(* IEC 61131-3 sources: Word/plc-course/12-data-structures/labs/starter, 3 files *)

(* ---- 12-1-recipe-manager.st ---- *)
(* Lab 12-1: Recipe manager - an array of structures, validated before use.
   Module 12 (Data structures). STARTER - the types, the recipe book, the
   limits and the program interface are declared for you. Write:
     1. the live check of the selected slot (SelectedOk),
     2. the load command: validate, then copy the whole recipe into Active,
        or reject it with the right LoadResult and change nothing.
   A FUNCTION for the value checks is a good idea (see the hint in the README).
   Then run:
     python3 tools/plctest.py 12-data-structures/labs/starter/12-1-recipe-manager.st *)

TYPE
  ST_Recipe :
  STRUCT
    Name    : STRING;               (* product name shown on the HMI; '' = empty slot *)
    Dose    : ARRAY[1..3] OF REAL;  (* kg of ingredient 1 (water), 2 (base), 3 (seasoning) *)
    Temp    : REAL;                 (* degC, batch temperature setpoint *)
    MixTime : TIME;                 (* mixing time once the batch is at temperature *)
  END_STRUCT;

  ST_RecipeLimits :
  STRUCT
    DoseMax    : REAL;              (* kg, largest dose of any one ingredient *)
    TotalMax   : REAL;              (* kg, vessel working capacity *)
    TempMin    : REAL;              (* degC *)
    TempMax    : REAL;              (* degC *)
    MixTimeMin : TIME;
    MixTimeMax : TIME;
  END_STRUCT;

  (* Result of the last load command. The first value is the initial value. *)
  E_LoadResult : (NotLoaded, Loaded, BadIndex, EmptySlot, BadValue, BatchBusy);
END_TYPE

PROGRAM RecipeManager
  VAR (* recipe book, edited on the HMI recipe screen. Slot 4 holds a typing
         mistake (95 degC) and slot 5 is empty, so both must be refused. *)
    Recipes : ARRAY[1..5] OF ST_Recipe := [
      (Name := 'Tomato soup',     Dose := [400.0, 150.0, 20.0], Temp := 85.0, MixTime := T#20m),
      (Name := 'Vegetable stock', Dose := [450.0, 300.0, 10.0], Temp := 80.0, MixTime := T#30m),
      (Name := 'Cheese sauce',    Dose := [250.0, 200.0, 50.0], Temp := 65.0, MixTime := T#15m),
      (Name := 'Trial batch',     Dose := [100.0, 100.0, 0.0],  Temp := 95.0, MixTime := T#10m)];
  END_VAR
  VAR (* HMI selection and command, and the state of the batch *)
    SelectNo     : INT;             (* recipe number chosen on the HMI; 0 = none *)
    LoadCmd      : BOOL;            (* HMI sets it to request a load; the PLC clears it *)
    BatchRunning : BOOL;            (* TRUE while a batch is in progress (from the sequence) *)
  END_VAR
  VAR (* results - keep these names *)
    SelectedOk   : BOOL;            (* the selected recipe could be loaded (enables the Load button) *)
    Active       : ST_Recipe;       (* the recipe the batch sequence uses *)
    ActiveNo     : INT;             (* which slot Active came from; 0 = nothing loaded yet *)
    LoadResult   : E_LoadResult;    (* outcome of the last load command *)
  END_VAR
  VAR CONSTANT
    RECIPE_LIMITS : ST_RecipeLimits := (DoseMax := 500.0, TotalMax := 1000.0,
                                        TempMin := 20.0, TempMax := 85.0,
                                        MixTimeMin := T#1m, MixTimeMax := T#2h);
    FIRST_SLOT : INT := 1;          (* keep in step with the ARRAY[1..5] bounds *)
    LAST_SLOT  : INT := 5;
  END_VAR
  (* TODO: add a VAR ... END_VAR block here for your internal variables. *)

  (* TODO: replace these placeholder lines with the recipe manager logic.
     Test the index BEFORE you read Recipes[SelectNo]. *)
  SelectedOk := FALSE;
  LoadCmd := FALSE;
END_PROGRAM

CONFIGURATION Config0
  RESOURCE Res0 ON PLC
    TASK MainTask(INTERVAL := T#10ms, PRIORITY := 0);
    PROGRAM Inst0 WITH MainTask : RecipeManager;
  END_RESOURCE
END_CONFIGURATION

(* ---- 12-2-event-log.st ---- *)
(* Lab 12-2: Event log - a ring buffer of structures.
   Module 12 (Data structures). STARTER - the event structure, the program
   interface and the millisecond clock are done for you.
   A pump station keeps its last ten events (code + time stamp) in a ring
   buffer: slots EventLog[0..9] are filled in turn, and when all ten are in
   use each new event overwrites the oldest. Entries never move. Write:
     1. the clear command,
     2. logging: one event per request into the next slot of the ring,
        overwriting the oldest entry when the log is full,
     3. the View outputs for the HMI.
   Then run:
     python3 tools/plctest.py 12-data-structures/labs/starter/12-2-event-log.st *)

TYPE
  ST_Event :
  STRUCT
    Code  : INT;    (* event code, 1..32767; 0 = empty entry *)
    Stamp : DINT;   (* ms since power-up when the event was logged *)
  END_STRUCT;
END_TYPE

PROGRAM EventLogger
  VAR (* requests from the rest of the program and the HMI *)
    NewCode  : INT;                      (* code of the event to log *)
    LogReq   : BOOL;                     (* TRUE = log NewCode now; the logger clears it *)
    ClearCmd : BOOL;                     (* TRUE = empty the log; the logger clears it *)
    ViewAge  : INT;                      (* HMI: 0 = newest event, 1 = the one before, ... *)
  END_VAR
  VAR (* the log - keep these names *)
    EventLog : ARRAY[0..9] OF ST_Event;  (* the ring: ten fixed slots *)
    Newest   : INT;                      (* slot of the newest entry (0 while the log is empty) *)
    Count    : INT;                      (* valid entries, 0..10 *)
    Total    : DINT;                     (* events logged since power-up or the last clear *)
    View     : ST_Event;                 (* the event ViewAge events back from the newest *)
    ViewValid : BOOL;                    (* TRUE when View holds a real event *)
  END_VAR
  VAR (* clock - given, do not change *)
    UpTime   : TON;
    NowMs    : DINT;                     (* ms since power-up *)
  END_VAR
  VAR CONSTANT
    LOG_SIZE : INT := 10;                (* keep in step with ARRAY[0..9] *)
    NO_EVENT : ST_Event := (Code := 0, Stamp := 0);
  END_VAR
  (* TODO: add a VAR ... END_VAR block here for your internal variables. *)

  (* ---- 0. Millisecond clock (given). TIME_TO_LREAL gives seconds in
     MATIEC and milliseconds in CODESYS; dividing by TIME_TO_LREAL(T#1s)
     gives seconds on both, and * 1000.0 makes milliseconds. The TON's ET
     stops at PT, so this clock is good for 24 days: fine for a lab. ---- *)
  UpTime(IN := TRUE, PT := T#24d);
  NowMs := LREAL_TO_DINT(TIME_TO_LREAL(UpTime.ET) / TIME_TO_LREAL(T#1s) * 1000.0);

  (* TODO: replace these placeholder lines with the clear, log and view logic.
     The HMI sets LogReq and ClearCmd; your logic clears them. *)
  LogReq := FALSE;
  ViewValid := FALSE;
END_PROGRAM

CONFIGURATION Config0
  RESOURCE Res0 ON PLC
    TASK MainTask(INTERVAL := T#10ms, PRIORITY := 0);
    PROGRAM Inst0 WITH MainTask : EventLogger;
  END_RESOURCE
END_CONFIGURATION

(* ---- 12-3-motor-array.st ---- *)
(* Lab 12-3: Four pumps, one data model, one loop.
   Module 12 (Data structures). STARTER - the data model (types), the
   program I/O, the array of pumps and the millisecond clock are done for you.
   MATIEC has no arrays of FB instances and no FB instances inside a STRUCT,
   so everything a pump must remember lives in its ST_MotorData element.
   Write:
     1. the input mapping (feedback inputs into Motors[i].RunFb),
     2. the pump logic for all four pumps in ONE FOR loop - in the program
        body, or in one FUNCTION_BLOCK instance that loops over the array,
     3. RunningCount and the output mapping (contactors, fault lamp).
   You may add members to the types (tests only use the documented ones).
   Then run:
     python3 tools/plctest.py 12-data-structures/labs/starter/12-3-motor-array.st

   Training exercise: the area stop here is an ordinary control stop, not an
   emergency stop. Emergency stops belong in a safety system (Module 20). *)

TYPE
  E_MotorState : (Stopped, Starting, Running, Faulted);

  ST_MotorCmd :
  STRUCT                          (* HMI -> PLC. The HMI sets a bit; the PLC clears it. *)
    Start : BOOL;
    Stop  : BOOL;
    Reset : BOOL;                 (* clears latched alarms; never starts the pump *)
  END_STRUCT;

  ST_MotorCfg :
  STRUCT                          (* engineer settings (retentive and change-controlled on a real plant) *)
    FbTimeoutMs : DINT := 2000;   (* ms that command and feedback may disagree *)
  END_STRUCT;

  ST_MotorSts :
  STRUCT                          (* PLC -> HMI, written by the PLC every scan *)
    State  : E_MotorState;
    RunCmd : BOOL;                (* command to the contactor *)
    Starts : DINT;                (* successful starts (Starting -> Running) since power-up *)
  END_STRUCT;

  ST_MotorAlm :
  STRUCT                          (* PLC -> HMI, latched until Reset *)
    FailToStart : BOOL;           (* started, but no feedback within FbTimeoutMs *)
    FbLost      : BOOL;           (* was running, feedback gone for FbTimeoutMs *)
    Uncommanded : BOOL;           (* stopped, but feedback present for FbTimeoutMs *)
  END_STRUCT;

  ST_MotorData :
  STRUCT
    Cmd        : ST_MotorCmd;
    Cfg        : ST_MotorCfg;
    Sts        : ST_MotorSts;
    Alm        : ST_MotorAlm;
    RunFb      : BOOL;            (* run feedback, copied from the input by the mapping layer *)
    DisagreeMs : DINT;            (* internal: ms that RunCmd and RunFb have disagreed *)
  END_STRUCT;
END_TYPE

PROGRAM FeedPumps
  VAR (* physical inputs *)
    P101_RunFb AT %IX0.0 : BOOL;          (* P-101 contactor auxiliary contact *)
    P102_RunFb AT %IX0.1 : BOOL;          (* P-102 contactor auxiliary contact *)
    P103_RunFb AT %IX0.2 : BOOL;          (* P-103 contactor auxiliary contact *)
    P104_RunFb AT %IX0.3 : BOOL;          (* P-104 discharge flow switch (slow to make) *)
    StopAll_NC AT %IX1.0 : BOOL;          (* area stop push-button, NC: TRUE = healthy *)
  END_VAR
  VAR (* physical outputs *)
    P101_Contactor AT %QX0.0 : BOOL;
    P102_Contactor AT %QX0.1 : BOOL;
    P103_Contactor AT %QX0.2 : BOOL;
    P104_Contactor AT %QX0.3 : BOOL;
    FaultLamp      AT %QX0.4 : BOOL;      (* ON while any pump is faulted *)
  END_VAR
  VAR (* the data model: one element per pump, read and written by the HMI *)
    Motors : ARRAY[1..4] OF ST_MotorData := [3((Cfg := (FbTimeoutMs := 2000))),
                                              (Cfg := (FbTimeoutMs := 5000))];
    RunningCount : INT;                   (* pumps proven running *)
  END_VAR
  VAR (* clock - given, do not change *)
    UpTime : TON;
    NowMs  : DINT;                        (* ms since power-up *)
  END_VAR
  (* TODO: add a VAR ... END_VAR block here for your internal variables. *)

  (* ---- Millisecond clock (given): ms since power-up. See Lab 12-2. ---- *)
  UpTime(IN := TRUE, PT := T#24d);
  NowMs := LREAL_TO_DINT(TIME_TO_LREAL(UpTime.ET) / TIME_TO_LREAL(T#1s) * 1000.0);

  (* TODO: replace these placeholder lines with the input mapping, the loop
     over Motors[1..4], RunningCount and the output mapping. *)
  P101_Contactor := FALSE;
  RunningCount := 0;
END_PROGRAM

CONFIGURATION Config0
  RESOURCE Res0 ON PLC
    TASK MainTask(INTERVAL := T#10ms, PRIORITY := 0);
    PROGRAM Inst0 WITH MainTask : FeedPumps;
  END_RESOURCE
END_CONFIGURATION
